TYPE ST_Filter_Current_Hexapod_Robot_Output :
STRUCT
	Current_Monitor: matrix_18_real_T;
END_STRUCT
END_TYPE

(* stored: Version 1.1.0.1, ProductVersion 3.1.4020.12
   DUT ST_Filter_Current_Hexapod_Robot_Output: Id {5ff930fa-b987-4f08-94d5-1c11cd46f543} *)
